TYPE TcaCarrierData :
STRUCT	
	Enabled : BOOL;
	Id : INT;
	Logging : WSTRING;	// Information in csv, xml or json Format
	Error : BOOL;	
	
	InitialStatus : eTcaWorkpiecePlaceStatus;
	RequestStatus : eTcaWorkpiecePlaceStatus;	

	WorkpiecesEnabled : ARRAY[0..TcaCarrier.MAX_WORKPIECEPLACES] OF BOOL;
	WorkpiecesCoordinate : ARRAY[0..TcaCarrier.MAX_WORKPIECEPLACES] OF ST_Coordinate;
	WorkpiecesData : ARRAY[0..TcaCarrier.MAX_WORKPIECEPLACES] OF TcaWorkpiecePlaceData;
	

END_STRUCT
END_TYPE

(* stored: Version 1.1.0.1
   DUT TcaCarrierData: Id {7f561e39-db64-406d-92fe-c6dddfbcdc12} *)
